PROGRAM StructuresAndFunctions
VAR
	myStruct : MyStruct;
	
	age : INT;
	name : STRING;
END_VAR

age := myStruct.age;
name := myStruct.name;

END_PROGRAM

(* stored: Version 1.1.0.1, ProductVersion 3.1.4024.11
   POU StructuresAndFunctions: Id {06824988-815b-4742-af74-335ba82413f9}, SpecialFunc None *)
